PROGRAM MAIN
VAR
	{attribute 'OPC.UA.DA':='1'}
	time_info:	FB_TIME;
END_VAR

time_info();

END_PROGRAM

(* stored: Version 1.1.0.1, ProductVersion 3.1.4024.3
   POU MAIN: Id {8c7f3494-d62b-4dce-8edb-a017c884dc00}, SpecialFunc None *)
